PROGRAM ExtMode_Init
VAR
	iSTEP : INT:= 0;
	Pulse1			: TP;
	Pulse2			: TP;
	Pulse3			: TP;
	Pulse4			: TP;
END_VAR


CASE iSTEP OF
	
	//KUKA ext init cmd
	0:	IF IO_KUKA.Init_Cmd OR IO.bButton THEN
			iSTEP := iSTEP + 1;
		END_IF
	
	//hardware toggle extmode n stopmess ON, then on move_enable n driveoff
	//then ON drive on
	1:	IF IO_KUKA.bEXT_mode THEN
			IO_KUKA.Init_Cmd := FALSE;
			IO_control.bMove_enable := IO_control.bDrive_off := TRUE;
			iSTEP := iSTEP + 1;
//		ELSE
//			IO_KUKA.Init_Cmd := FALSE;
//			iSTEP := 0;
		END_IF
		
	2:	IF IO_control.bMove_enable THEN
			IO_control.bIO_Act := TRUE;
			IO_control.bDrive_on := TRUE;
			IO_KUKA.Init_Cmd := FALSE;
			iSTEP := iSTEP + 1;
		END_IF	
	
	//if peri_ready on, then off drive_on
	3:	IF IO_KUKA.bPeri_ready THEN
			IO_control.bDrive_on := FALSE;
			iSTEP := iSTEP + 1;
		ELSE
			iSTEP := 0;
		END_IF
	
	//IF drive_on is ON, ON conf_mess, then if stopmess is OFF, OFF confmess
	4:	IF IO_control.bDrive_on = FALSE THEN
			IO_control.bConf_msg := TRUE;
			IF NOT IO_KUKA.bStopmess THEN
				IO_control.bConf_msg := FALSE;
				iSTEP := iSTEP + 1;
			ELSE
				iSTEP := 0;
			END_IF
		ELSE
			IO_KUKA.Init_Cmd := FALSE;
			iSTEP := 0;
		END_IF
	
	//confmess OFF, ON ext_start, when pro_act is OFF, off ext_start	
	5:	IF IO_control.bConf_msg = FALSE THEN
			IO_KUKA.bExt_start := TRUE;
			iSTEP := iSTEP + 1;
		ELSE
			iSTEP := 0;
		END_IF
		
	6:	IF IO_KUKA.bPro_act THEN
			IO_control.bExt_start := FALSE;		
			iSTEP := 0;
		ELSE
			iSTEP := 0;
		END_IF	
		
		
END_CASE

END_PROGRAM

(* stored: Version 1.1.0.1, ProductVersion 3.1.4024.12
   POU ExtMode_Init: Id {208ca540-6b2a-4ae5-84e7-ac901ada21d3}, SpecialFunc None *)
